INTERFACE IExpression EXTENDS __System.IQueryInterface

METHOD IsTrue : BOOL
VAR_INPUT
	i_ptrProcessState: POINTER TO ProcessState;
END_VAR
END_METHOD

METHOD ToString : STRING(256)
VAR_INPUT
END_VAR
END_METHOD

END_INTERFACE

(* stored: Version 1.1.0.1, ProductVersion 3.1.4024.12
   Itf IExpression: Id {c727e5ae-f079-4e5b-b922-afaa62c9fe0e}
   Method IsTrue: Id {d55e8b23-d898-426b-80c6-7c0f54d09339}
   Method ToString: Id {5ecdd8c1-0284-443e-8771-8bd768be6ce6} *)
